FUNCTION transpose : BOOL
VAR_IN_OUT
	a,att:ARRAY[*,*] OF LREAL;
END_VAR
VAR_INPUT
	m,n:SINT;
END_VAR
VAR
	i,j:SINT;
END_VAR


    FOR i:=0 TO m-1 DO 
        FOR j:=0 TO n-1 DO 
            att[j,i] := a[i,j];
        END_FOR
	END_FOR
	transpose:=true;

END_FUNCTION

(* stored: Version 1.1.0.1, ProductVersion 3.1.4024.12
   POU transpose: Id {c5ce8849-9b23-4721-a64c-567b73b2f772}, SpecialFunc None *)
